// TwinCAT 3 PLC project MBIDivB
// Title: Experiment Control Library
// Company: MBI DIv-B
// Author: Michael Schneider
// ProjectVersion: 0.1.0.0
// Description: Collection of function blocks used for data acquisition and experiment control.
// ProgramVersion: 3.1.4024.0
// libraries:
//   Tc2_Standard, * (Beckhoff Automation GmbH)
//   Tc2_System, * (Beckhoff Automation GmbH)
//   Tc3_Module, * (Beckhoff Automation GmbH)
// project tree:
//   DUTs/ CounterState.TcDUT, TriggerState.TcDUT
//   GVLs/ globals.TcGVL
//   / PlcTask.TcTTO
//   POUs/ AnalogInput.TcPOU, AnalogOutput.TcPOU, CounterTimer.TcPOU, FilterRingBuffer.TcPOU, MultiTrigger.TcPOU, getTaskCycleTime.TcPOU, RampCtrl.TcPOU, ReedFlowMeter.TcPOU
//   Version/ Global_Version.TcGVL
// real-time tasks:
//   TASK PlcTask: cycle T#10ms, priority 20, ADS port 350

CONFIGURATION MBIDivB
    RESOURCE PLC ON TwinCAT3
        TASK PlcTask(INTERVAL := T#10ms, PRIORITY := 20);
        PROGRAM MAIN WITH PlcTask : MAIN;
    END_RESOURCE
END_CONFIGURATION

// ---- DUTs/CounterState.TcDUT
{attribute 'qualified_only'}
{attribute 'strict'}
TYPE CounterState :
(
	STOP, MEASURE, WAIT
);
END_TYPE

// ---- DUTs/TriggerState.TcDUT
{attribute 'qualified_only'}
{attribute 'strict'}
TYPE TriggerState :
(
	STOPPED, DELAY, ACTIVE_LOW, ACTIVE_HIGH
);
END_TYPE

// ---- GVLs/globals.TcGVL
{attribute 'qualified_only'}
VAR_GLOBAL CONSTANT
	MAX_BUFFER_LENGTH: UDINT := 100_000;
END_VAR

// ---- Version/Global_Version.TcGVL
{attribute 'TcGenerated'}
{attribute 'no-analysis'}
{attribute 'linkalways'}
// This function has been automatically generated from the project information.
VAR_GLOBAL CONSTANT
	{attribute 'const_non_replaced'}
	stLibVersion_Experiment_Control_Library : ST_LibVersion := (iMajor := 0, iMinor := 1, iBuild := 0, iRevision := 0, nFlags := 0, sVersion := '0.1.0.0');
END_VAR

// ---- POUs/AnalogInput.TcPOU
FUNCTION_BLOCK AnalogInput
VAR
	nMaxRawValue: DINT := 7812500;  // for 24 bit device, e.g. ELM300x - check manual
	nRawValue AT %I*: DINT; // signed 32 bit integer representing full value range
	fMaxVoltage: REAL := 10; // measurement range
	valuebuffer: CounterTimer; // buffer for timed measurements
	filterbuffer: FilterRingBuffer;
	nFilterSize: UDINT := 100;
	fVoltage: REAL;
	fVoltageFiltered: REAL; // running average filter
END_VAR

fVoltage := fMaxVoltage * DINT_TO_REAL(nRawValue) / DINT_TO_REAL(nMaxRawValue);  

IF filterbuffer.nBufferSize <> nFilterSize THEN
	nFilterSize := filterbuffer.SetFilterSize(nFilterSize);
END_IF
filterbuffer.Store(fVoltage);
fVoltageFiltered := filterbuffer.CalculateMean();

valuebuffer(fValue:=fVoltage);  // makes sure buffer in initialized and calls StoreValueConditional

END_FUNCTION_BLOCK

// ---- POUs/CounterTimer.TcPOU
FUNCTION_BLOCK CounterTimer
VAR_INPUT
	fValue : REAL;
END_VAR
VAR
	values: ARRAY[0 .. globals.MAX_BUFFER_LENGTH] OF REAL;
	fValueSum: REAL := 0;
	fValueAverage: REAL := 0;
	
	nScanTotal: UDINT := 1;
	nLatencyCycles: UDINT := 0;
	nAccumCycles: UDINT := 100;
	
	nScanIndex: UDINT := 0;
	nWaitIndex: UDINT := 0;
	nAccumIndex: UDINT := 0;
	
	eState: CounterState:=CounterState.STOP;
	nState: INT; // for pyads, since it can't read the enum value properly
END_VAR

// Value counter and buffer. Performs consecutive measurements with
// configurable integration time and delay between measurements.

ProcessValue(fValue);
nState := eState;

METHOD PrepareMeasurement
VAR_INPUT
	nAccumMilliseconds: UDINT;
	nDelayMilliseconds: UDINT;
	nMeasurements: UDINT;
END_VAR
VAR
	nCyclesPerMillisecond: UDINT;
END_VAR
// CycleTime is in multiples of 100 ns
nCyclesPerMillisecond := 10_000 / getTaskCycleTime();

nScanTotal := LIMIT(1, nMeasurements, globals.MAX_BUFFER_LENGTH);
nAccumCycles := MAX(1, nAccumMilliseconds * nCyclesPerMillisecond);
nLatencyCycles := nDelayMilliseconds * nCyclesPerMillisecond;
END_METHOD

METHOD ProcessValue
VAR_INPUT
	fValue : REAL;
END_VAR
// integrate values for given number of ticks, then store average
// enter wait loop after storing

IF eState = CounterState.MEASURE THEN
	fValueSum := fValueSum + fValue;
	nAccumIndex := nAccumIndex + 1;
	fValueAverage := fValueSum / UDINT_TO_REAL(nAccumIndex);

	IF nAccumIndex >= nAccumCycles THEN
		values[nScanIndex] := fValueAverage;
		nScanIndex := nScanIndex + 1;
		nAccumIndex := 0;
		fValueSum := 0;
		
		IF nScanIndex >= nScanTotal THEN
			eState := CounterState.STOP;
		ELSE
			eState := CounterState.WAIT;
			nWaitIndex := 0;	
		END_IF
	END_IF
END_IF

IF eState = CounterState.WAIT THEN
	IF nWaitIndex >= nLatencyCycles THEN
		eState := CounterState.MEASURE;			
	ELSE
		nWaitIndex := nWaitIndex + 1;
	END_IF
END_IF
END_METHOD

METHOD StartBuffer
eState := CounterState.MEASURE;
nScanIndex := 0;
nWaitIndex := 0;
nAccumIndex := 0;
fValueSum := 0;
END_METHOD

METHOD StopBuffer
eState := CounterState.STOP;
END_METHOD

END_FUNCTION_BLOCK

// ---- POUs/getTaskCycleTime.TcPOU
FUNCTION getTaskCycleTime : UDINT  // return cycle time in integer multiples of 100 ns
VAR_INPUT
END_VAR
VAR
END_VAR

getTaskCycleTime := TwinCAT_SystemInfoVarList._TaskInfo[GETCURTASKINDEXEX()].CycleTime;

END_FUNCTION

// ---- POUs/FilterRingBuffer.TcPOU
FUNCTION_BLOCK FilterRingBuffer
VAR CONSTANT
	MAX_BUFFER_SIZE: UDINT := 1000;
END_VAR
VAR_OUTPUT
	fRunningAverage: REAL;
END_VAR
VAR
	buffer: ARRAY [0 .. MAX_BUFFER_SIZE] OF REAL;
	nBufferSize: UDINT := 100;
	nCurrentIndex: UDINT := 0;
	nValidEntries: UDINT := 0;
END_VAR


fRunningAverage := CalculateMean();

METHOD CalculateMean : REAL

VAR
	n: UDINT;
END_VAR
CalculateMean := 0;
FOR n := 0 TO nValidEntries DO
	CalculateMean := CalculateMean + buffer[n];
END_FOR

CalculateMean := CalculateMean / UDINT_TO_REAL(nValidEntries);
END_METHOD

METHOD SetFilterSize
VAR_INPUT
	nFilterSize: UDINT;
END_VAR
VAR_OUTPUT
	nNewFilterSize: UDINT;
END_VAR
nBufferSize := MAX(1, MIN(nFilterSize, MAX_BUFFER_SIZE));
nCurrentIndex := 0;
nValidEntries := 0;
nNewFilterSize := nBufferSize;
END_METHOD

METHOD Store
VAR_INPUT
	fValue: REAL;
END_VAR
buffer[nCurrentIndex] := fValue;
nCurrentIndex := (nCurrentIndex + 1) MOD nBufferSize;
nValidEntries := MIN(nValidEntries + 1, nBufferSize);
END_METHOD

END_FUNCTION_BLOCK

// ---- POUs/AnalogOutput.TcPOU
(*
:Description: Control analog output with a linear ramp.
:Usage: Just call in MAIN loop. Internal parameters are intended to be set by ADS.
:Relevant ADS Symbols:
- Setpoint: the target value (rw)
- RawScale: Conversion factor between voltage and raw value (default: 32768/10)
- LimitMin: Minimum voltage allowed
- LimitMax: Maximum voltage allowed
- Ramp.MomentarySetpoint: the current output value (ro)
- Ramp.SetpointReached: whether the ramp is finished or not
- Ramp.Velocity: ramp speed in V/s
*)

FUNCTION_BLOCK AnalogOutput
VAR
	RawOutput AT %Q*: INT;
	RawScale: REAL := 32768 / 10;
	Setpoint: REAL := 0;
	LimitMin: REAL := -10;
	LimitMax: REAL := 10;
	Ramp: RampCtrl;
END_VAR

Setpoint := LIMIT(Setpoint, LimitMin, LimitMax);
Ramp(Target:=Setpoint);
RawOutput := REAL_TO_INT(RawScale * Ramp.MomentarySetpoint);

END_FUNCTION_BLOCK

// ---- POUs/RampCtrl.TcPOU
FUNCTION_BLOCK RampCtrl
VAR_INPUT
	Target: REAL := 0;
END_VAR
VAR_OUTPUT
	MomentarySetpoint: REAL := 0;
END_VAR
VAR
	Initialized: BOOL := FALSE;
	Velocity: REAL := 1;
	CycleTimeSeconds: REAL := 0;
	Direction: REAL;
	SetpointReached: BOOL := FALSE;
END_VAR

IF NOT Initialized THEN  // initialization
	CycleTimeSeconds := UDINT_TO_REAL(getTaskCycleTime()) / 10_000_000;
	Initialized := TRUE;
END_IF

SetpointReached := (Target = MomentarySetpoint);

IF NOT SetpointReached THEN
	Direction := (Target - MomentarySetpoint) / ABS(Target - MomentarySetpoint);
	MomentarySetpoint := MomentarySetpoint + Direction * Velocity * CycleTimeSeconds;
	IF Direction < 0 THEN
		MomentarySetpoint := MAX(Target, MomentarySetpoint);
	ELSE
		MomentarySetpoint := MIN(Target, MomentarySetpoint);
	END_IF
END_IF

END_FUNCTION_BLOCK

// ---- POUs/MultiTrigger.TcPOU
FUNCTION_BLOCK MultiTrigger
VAR
	Output AT %Q*: BOOL;
	Start: BOOL := FALSE;
	Active: BOOL := FALSE;
	State: TriggerState := TriggerState.STOPPED;
	TicksDelay: UINT := 0;
	TicksHigh: UINT := 100;
	TicksLow: UINT := 100;
	NumTrigger: INT := 20;
	NumCurrent: INT := 0;
	TickCount: UINT := 0;
	Stop: BOOL := FALSE;
END_VAR

TicksHigh := MAX(1, TicksHigh);
TicksLow := MAX(1, TicksLow);

TickCount := TickCount + 1;

IF Start THEN
	Start := FALSE;
	startTrigger();
END_IF

IF Stop THEN
	Stop := FALSE;
	setState(Target:=TriggerState.STOPPED);
END_IF

CASE State OF
	TriggerState.DELAY:
		IF TickCount >= TicksDelay THEN
			setState(Target:=TriggerState.ACTIVE_HIGH);
		END_IF
		
	TriggerState.ACTIVE_HIGH:
		IF TickCount >= TicksHigh THEN
			IF NumCurrent = NumTrigger THEN
				setState(Target:=TriggerState.STOPPED);
			ELSE
				setState(Target:=TriggerState.ACTIVE_LOW);
			END_IF
		END_IF
		
	TriggerState.ACTIVE_LOW:
		IF TickCount >= TicksLow THEN
			NumCurrent := NumCurrent + 1;
			setState(Target:=TriggerState.ACTIVE_HIGH);
		END_IF
END_CASE

METHOD setState
VAR_INPUT
	Target: TriggerState;
END_VAR
CASE Target OF
	TriggerState.STOPPED:
		Output := FALSE;
		Active := FALSE;
		State := TriggerState.STOPPED;
	TriggerState.DELAY:
		Output := FALSE;
		Active := TRUE;
		State := TriggerState.DELAY;
	TriggerState.ACTIVE_HIGH:
		Output := TRUE;
		Active := TRUE;
		State := TriggerState.ACTIVE_HIGH;
	TriggerState.ACTIVE_LOW:
		Output := FALSE;
		Active := TRUE;
		State := TriggerState.ACTIVE_LOW; 
END_CASE

TickCount := 0;
END_METHOD

(*
:Description: Public method to start trigger in case setting Start attribute directly is not possible.
*)
METHOD PUBLIC startTrigger
VAR_INPUT
END_VAR
NumCurrent := 0;
IF TicksDelay > 0 THEN
	setState(Target:=TriggerState.DELAY);
ELSE
	setState(Target:=TriggerState.ACTIVE_HIGH);
END_IF
END_METHOD

END_FUNCTION_BLOCK

// ---- POUs/ReedFlowMeter.TcPOU
FUNCTION_BLOCK ReedFlowMeter
VAR CONSTANT
	MAXLEN: UINT := 1000;
	TIMEUNITSPERSECOND: LINT := 10_000_000; // 100 ns per step
END_VAR
VAR
	fFrequencyToFlowScale: REAL := 0.28;
	fFlowRate: REAL;
	bReedSwitch AT %I*: BOOL;
	nIndex: UINT;
	timestamps: ARRAY [0..MAXLEN] OF ULINT;
	nTimeNow: ULINT; // 100 ns per unit
	nTriggerCount: UINT;
	nLoopIndex: UINT;
	trigger: R_TRIG;
END_VAR

// Koolance INS-FM19 flow meter
// simple reed contact switch
// frequency directly proportional to flow rate
// typical frequencies are <30 Hz, so no fast counter required

nTimeNow := F_GetSystemTime();
trigger(CLK:=bReedSwitch);
IF trigger.Q THEN
	timestamps[nIndex] := nTimeNow;
	nIndex := (nIndex + 1) MOD  MAXLEN;
END_IF

nTriggerCount := 0;
FOR nLoopIndex := 0 TO MAXLEN DO
	IF (ULINT_TO_LINT(nTimeNow) - ULINT_TO_LINT(timestamps[nLoopIndex])) < TIMEUNITSPERSECOND THEN
		nTriggerCount := nTriggerCount + 1;
	END_IF
END_FOR

fFlowRate := fFrequencyToFlowScale * nTriggerCount;

END_FUNCTION_BLOCK
